FUNCTION_BLOCK DelayOnAndTrue (* Extracted Composite Function Block Type *)
  (* Standard: 61499-2 *)
  (* Version 10/14/2024, 2001a *)
  PACKAGE Main;
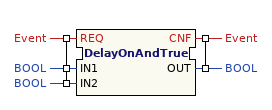
  EVENT_INPUT
    REQ WITH IN1, IN2; (* Normal Execution Request *)
  END_EVENT
  EVENT_OUTPUT
    CNF WITH OUT;
  END_EVENT
  VAR_INPUT
    IN1 : BOOL; (* Argument *)
    IN2 : BOOL; (* Argument *)
  END_VAR
  VAR_OUTPUT
    OUT : BOOL; (* Result: IN1 AND IN2 AND ... *)
  END_VAR
  FBS
    FB8 : AND_88A3DD8EC65DD11C; {SET_ATTRIBUTE(Configuration.GenericFBType.InterfaceParams, Runtime.Standard#CNT:=2;OUT:BOOL)}
    FB3 : E_DELAY(DT := T#1000ms);
    FB1 : E_PERMIT;
    FB2 : NOT_42C76073DCEB1A7A; {SET_ATTRIBUTE(Configuration.GenericFBType.InterfaceParams, Runtime.Standard#CNT:=1;OUT${CNT$}:BOOL)}
    FB4 : E_PERMIT;
    FB5 : E_MERGE;
  END_FBS
  EVENT_CONNECTIONS
    REQ TO FB8.REQ;
    FB8.CNF TO FB2.REQ;
    FB2.CNF TO FB1.EI;
    FB1.EO TO FB3.STOP;
    FB8.CNF TO FB4.EI;
    FB4.EO TO FB3.START;
    FB3.EO TO FB5.EI1;
    FB1.EO TO FB5.EI2;
    FB5.EO TO CNF;
  END_CONNECTIONS
  DATA_CONNECTIONS
    IN1 TO FB8.IN1;
    IN2 TO FB8.IN2;
    FB8.OUT TO FB2.IN1;
    FB2.OUT1 TO FB1.PERMIT;
    FB8.OUT TO FB4.PERMIT;
    FB8.OUT TO OUT;
  END_CONNECTIONS
END_FUNCTION_BLOCK
